TcoUtilities.TcoDintToBytes(inFormat := TcoUtilities.eTcoDataFormat.LittleEndian,
    inValue := REAL_TO_DINT((_control.Coordinates.Rz + 360.0) * 10000.0),
    outByte0 := inoData.Out.Outputs[index],
    outByte1 := inoData.Out.Outputs[index + 1],
    outByte2 := inoData.Out.Outputs[index + 2],
    outByte3 := inoData.Out.Outputs[index + 3]);
END_METHOD

METHOD INTERNAL UpdateStatus
VAR
    _message : STRING(125);
    tempOut : BYTE;
    index : INT;
    _bytes : DINT;
END_VAR
//SYSTEM INPUTS
index := 0;
_status.State.AutoOn := inoData.In.Inputs[index].0;
_status.State.CycleOn := inoData.In.Inputs[index].1;
_status.State.EmgStop := inoData.In.Inputs[index].2;
_status.State.Error := inoData.In.Inputs[index].3;
_status.State.MoveActive := inoData.In.Inputs[index].4;
_status.State.MoveInactive := inoData.In.Inputs[index].5;
_status.State.MotorOff := inoData.In.Inputs[index].6;
_status.State.MotorOn := inoData.In.Inputs[index].7;
index := 1;
_status.State.MotorOffState := inoData.In.Inputs[index].0;
_status.State.MotorOnState := inoData.In.Inputs[index].1;
_status.State.ProgExecError := inoData.In.Inputs[index].2;
_status.State.SafetyOk := inoData.In.Inputs[index].3;
_status.State.SystemInputBusy := inoData.In.Inputs[index].4;
_status.State.PpMoved := inoData.In.Inputs[index].5;
_status.State.MotionSupervision := inoData.In.Inputs[index].6;
_status.State.BatteryLow := inoData.In.Inputs[index].7;
//Area/positions flags this  should be obsolete because Zones and InPosition is used as byte below
index := 2;
_status.State.InArea_1 := inoData.In.Inputs[index].0;
_status.State.InArea_2 := inoData.In.Inputs[index].1;
_status.State.InArea_3 := inoData.In.Inputs[index].2;
_status.State.InArea_4 := inoData.In.Inputs[index].3;
_status.State.InPosition_1 := inoData.In.Inputs[index].4;
_status.State.InPosition_2 := inoData.In.Inputs[index].5;
_status.State.InPosition_3 := inoData.In.Inputs[index].6;
_status.State.InPosition_4 := inoData.In.Inputs[index].7;
//
//Tool signals
index := 3;
_status.State.Tool_1_Retract := inoData.In.Inputs[index].0;
_status.State.Tool_1_Extend := inoData.In.Inputs[index].1;
_status.State.Tool_2_Retract := inoData.In.Inputs[index].2;
_status.State.Tool_2_Extend := inoData.In.Inputs[index].3;
_status.State.Tool_3_Retract := inoData.In.Inputs[index].4;
_status.State.Tool_3_Extend := inoData.In.Inputs[index].5;
_status.State.Tool_4_Retract := inoData.In.Inputs[index].6;
_status.State.Tool_4_Extend := inoData.In.Inputs[index].7;
//Safety signals
index := 4;
_status.State.AutoStop_1 := inoData.In.Inputs[index].0;
_status.State.AutoStop_2 := inoData.In.Inputs[index].1;
_status.State.EmergencyStop_1 := inoData.In.Inputs[index].2;
_status.State.EmergencyStop_2 := inoData.In.Inputs[index].3;
_status.State.GeneralStop_1 := inoData.In.Inputs[index].4;
_status.State.GeneralStop_2 := inoData.In.Inputs[index].5;
_status.State.Enable_1 := inoData.In.Inputs[index].6;
_status.State.Enable_2 := inoData.In.Inputs[index].7;
index := 5;
_status.State.Zone := inoData.In.Inputs[index];
index := 6;
_status.State.InPosition := inoData.In.Inputs[index];
//Movement parameters
index := 7;
_status.State.ActionNo := inoData.In.Inputs[index];
index := 8;
_status.State.GlobalSpeed := inoData.In.Inputs[index];
index := 9;
_status.State.ToolNo := inoData.In.Inputs[index];
index := 10;
_status.State.WorkobjectNo := inoData.In.Inputs[index];
index := 11;
_status.State.PointNo := inoData.In.Inputs[index];
index := 12;

_status.State.UserSpecSpeed1 := TcoUtilities.TcoBytesToDint(inFormat := TcoUtilities.eTcoDataFormat.LittleEndian,
    inByte0 := inoData.In.Inputs[index],
    inByte1 := inoData.In.Inputs[index + 1],
    inByte2 := inoData.In.Inputs[index + 2],
    inByte3 := inoData.In.Inputs[index + 3]);

index := 16;

_status.State.UserSpecSpeed2 := TcoUtilities.TcoBytesToDint(inFormat := TcoUtilities.eTcoDataFormat.LittleEndian,
    inByte0 := inoData.In.Inputs[index],
    inByte1 := inoData.In.Inputs[index + 1],
    inByte2 := inoData.In.Inputs[index + 2],
    inByte3 := inoData.In.Inputs[index + 3]);

index := 20;

_bytes := TcoUtilities.TcoBytesToDint(inFormat := TcoUtilities.eTcoDataFormat.LittleEndian,
    inByte0 := inoData.In.Inputs[index],
    inByte1 := inoData.In.Inputs[index + 1],
    inByte2 := inoData.In.Inputs[index + 2],
    inByte3 := inoData.In.Inputs[index + 3]);

_status.State.Coordinates.X := (DINT_TO_REAL(_bytes) / 10000.0) - 10000.0;
index := 24;

_bytes := TcoUtilities.TcoBytesToDint(inFormat := TcoUtilities.eTcoDataFormat.LittleEndian,
    inByte0 := inoData.In.Inputs[index],
    inByte1 := inoData.In.Inputs[index + 1],
    inByte2 := inoData.In.Inputs[index + 2],
    inByte3 := inoData.In.Inputs[index + 3]);

_status.State.Coordinates.Y := (DINT_TO_REAL(_bytes) / 10000.0) - 10000.0;
index := 28;

_bytes := TcoUtilities.TcoBytesToDint(inFormat := TcoUtilities.eTcoDataFormat.LittleEndian,
    inByte0 := inoData.In.Inputs[index],
    inByte1 := inoData.In.Inputs[index + 1],
    inByte2 := inoData.In.Inputs[index + 2],
    inByte3 := inoData.In.Inputs[index + 3]);

_status.State.Coordinates.Z := (DINT_TO_REAL(_bytes) / 10000.0) - 10000.0;
index := 32;

_bytes := TcoUtilities.TcoBytesToDint(inFormat := TcoUtilities.eTcoDataFormat.LittleEndian,
    inByte0 := inoData.In.Inputs[index],
    inByte1 := inoData.In.Inputs[index + 1],
    inByte2 := inoData.In.Inputs[index + 2],
    inByte3 := inoData.In.Inputs[index + 3]);

_status.State.Coordinates.Rx := (DINT_TO_REAL(_bytes) / 10000.0) - 360.0;
index := 36;

_bytes := TcoUtilities.TcoBytesToDint(inFormat := TcoUtilities.eTcoDataFormat.LittleEndian,
    inByte0 := inoData.In.Inputs[index],
    inByte1 := inoData.In.Inputs[index + 1],
    inByte2 := inoData.In.Inputs[index + 2],
    inByte3 := inoData.In.Inputs[index + 3]);

_status.State.Coordinates.Ry := (DINT_TO_REAL(_bytes) / 10000.0) - 360.0;
index := 40;

_bytes := TcoUtilities.TcoBytesToDint(inFormat := TcoUtilities.eTcoDataFormat.LittleEndian,
    inByte0 := inoData.In.Inputs[index],
    inByte1 := inoData.In.Inputs[index + 1],
    inByte2 := inoData.In.Inputs[index + 2],
    inByte3 := inoData.In.Inputs[index + 3]);

_status.State.Coordinates.Rz := (DINT_TO_REAL(_bytes) / 10000.0) - 360.0;
index := 44;

_status.State.EventId := TcoUtilities.TcoBytesToUDint(inFormat := TcoUtilities.eTcoDataFormat.LittleEndian,
    inByte0 := inoData.In.Inputs[index],
    inByte1 := inoData.In.Inputs[index + 1],
    inByte2 := inoData.In.Inputs[index + 2],
    inByte3 := inoData.In.Inputs[index + 3]);
END_METHOD

END_FUNCTION_BLOCK
